{attribute 'TcGenerated'}
{attribute 'no-analysis'}
{attribute 'linkalways'}
// This function has been automatically generated from the project information.
VAR_GLOBAL CONSTANT
	{attribute 'const_non_replaced'}
	stLibVersion_TwinCAT_Open_Framework_Collections : ST_LibVersion := (iMajor := 1, iMinor := 0, iBuild := 13, iRevision := 0, nFlags := 0, sVersion := '1.0.13.0');
END_VAR

(* stored: Version 1.1.0.1
   GVL Global_Version: Id {c1c88166-1a0b-4a85-9077-caff5f7e86e1} *)
